(* CoDeSys 2.3 export: PRG_MAIN.EXP *)

(* POU PRG_MAIN, SFC *)
PROGRAM PRG_MAIN
VAR
END_VAR
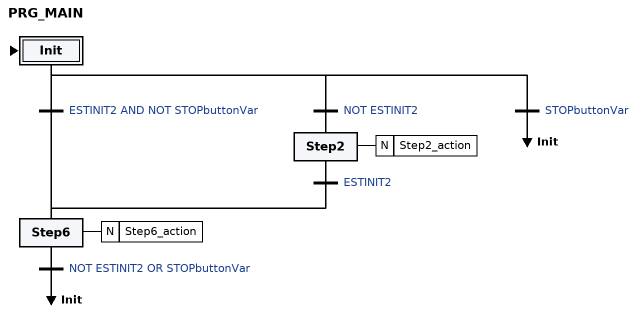
INITIAL_STEP Init:
END_STEP
TRANSITION FROM Init TO Step6 := ESTINIT2 AND NOT STOPbuttonVar;
END_TRANSITION
TRANSITION FROM Init TO Step2 := NOT ESTINIT2;
END_TRANSITION
TRANSITION FROM Init TO Init := STOPbuttonVar;
END_TRANSITION
STEP Step2:
	Step2_action(N);
END_STEP
TRANSITION FROM Step2 TO Step6 := ESTINIT2;
END_TRANSITION
STEP Step6:
	Step6_action(N);
END_STEP
TRANSITION FROM Step6 TO Init := NOT ESTINIT2 OR STOPbuttonVar;
END_TRANSITION

ACTION Step2_action:
IF StanbyActive THEN Correspondance_Etages ();END_IF
Initialisation_reset();
SENS_M:=TRUE;
END_ACTION

ACTION Step6_action:
PAL_COMMUN_ETAGE;
StandBY;
Clignotement;
STOP_PORTES();
Correspondance_Etages();
END_ACTION
END_PROGRAM
